// TIA Portal V15.1 export
// export: Created 2024-05-17T05:38:41.6843749Z, ExportSetting WithDefaults, DisplayName Totally Integrated Automation Portal, DisplayVersion V15.1 Update 5, DisplayName TIA Portal Openness, DisplayVersion V15.1 Update 5, DisplayName SINAMICS Startdrive Advanced, DisplayVersion V15.1, DisplayName G130, G150, S120, S150, SINAMICS MV, S210, DisplayVersion V15.1, DisplayName G110M, G120, G120C, G120D, G120P, DisplayVersion V15.1, DisplayName STEP 7 Professional, DisplayVersion V15.1 Update 5, DisplayName STEP 7 Safety, DisplayVersion V15.1, DisplayName WinCC Professional, DisplayVersion V15.1 Update 5, DisplayName SIMATIC Visualization Architect, DisplayVersion V15.1
FUNCTION "LGBHoist2Pos2S-FC302PN-Config" : Void   // FC6606, FBD
TITLE = LMoveEPos-Config / LHoist2Pos2S-FC302PN-Config
{ S7_Optimized_Access := 'FALSE' }
AUTHOR : VCC
FAMILY : Config
VERSION : 0.0.0.0
// =============================================================================
// Configuration MoveUnitEpos
// =============================================================================
// stored: AutoNumber false, IsIECCheckEnabled false, SetENOAutomatically False, UDAEnableTagReadback false
   VAR_INPUT
      C_InitDirection : Bool;   // Config
      C_SafetySwNc : Bool;   // Config
      C_SafetySwUsed : Bool;   // Config
      C_MotorProtectionNc : Bool;   // Config
      C_MotorProtectionUsed : Bool;   // Config
      C_BrakeProtectionNc : Bool;   // Config
      C_BrakeProtectionUsed : Bool;   // Config
      C_ReleaseBrakeUsed : Bool;   // Release brake used / Config
      C_MotionStopUsed : Bool;   // Config
      C_EnableAlarmHW : Bool;   // Enable Alarm hardware (e.g. safetyswitch, motorprotector, detections) / Config
      C_EnablePNReset : Bool;   // Config
      C_NotQuickStop : Bool;   // QuickStop function; When FALSE the QuickStop of the G120 is active / Config
      C_RunTimeMaxSetAlm : DInt;   // Maximum Time (x1ms) that the function may run (create Overtime) / Config
      C_RunTimeMaxResAlm : DInt;   // Maximum Time (x1ms) that the function may run (create Overtime) / Config
      C_HWSubInput : HW_SUBMODULE;   // I/O / Config
      C_HWSubOutput : HW_SUBMODULE;   // I/O / Config
   END_VAR
   VAR_IN_OUT
      IO_Config : "Hoist2Pos2S-FC302PNConfig";   // Output Word / Config
   END_VAR
BEGIN

REGION Network 1: **** 1 - Inputs **** Move Bit Config
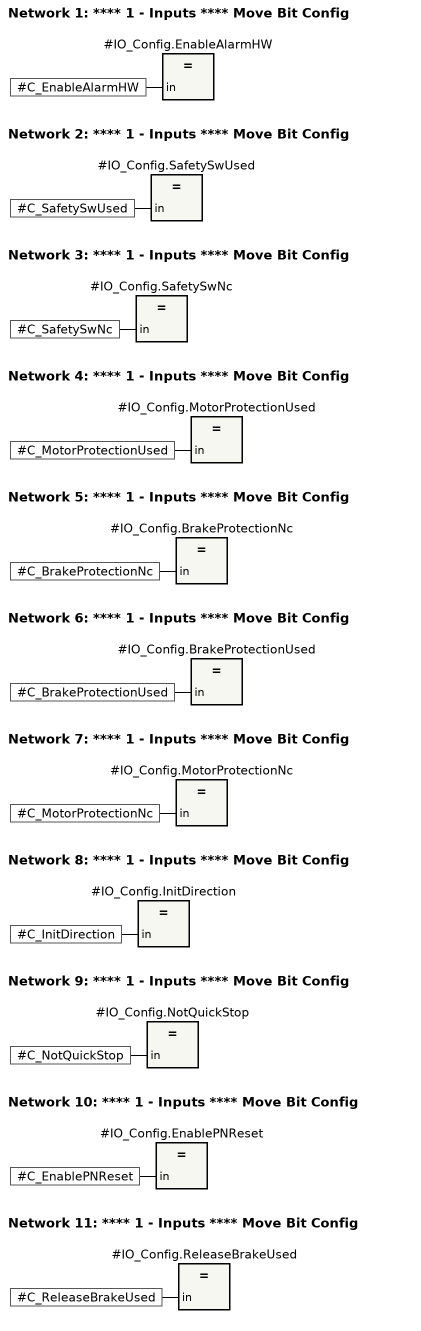
   #IO_Config.EnableAlarmHW := #C_EnableAlarmHW;
END_REGION

REGION Network 2: **** 1 - Inputs **** Move Bit Config
   #IO_Config.SafetySwUsed := #C_SafetySwUsed;
END_REGION

REGION Network 3: **** 1 - Inputs **** Move Bit Config
   #IO_Config.SafetySwNc := #C_SafetySwNc;
END_REGION

REGION Network 4: **** 1 - Inputs **** Move Bit Config
   #IO_Config.MotorProtectionUsed := #C_MotorProtectionUsed;
END_REGION

REGION Network 5: **** 1 - Inputs **** Move Bit Config
   #IO_Config.BrakeProtectionNc := #C_BrakeProtectionNc;
END_REGION

REGION Network 6: **** 1 - Inputs **** Move Bit Config
   #IO_Config.BrakeProtectionUsed := #C_BrakeProtectionUsed;
END_REGION

REGION Network 7: **** 1 - Inputs **** Move Bit Config
   #IO_Config.MotorProtectionNc := #C_MotorProtectionNc;
END_REGION

REGION Network 8: **** 1 - Inputs **** Move Bit Config
   #IO_Config.InitDirection := #C_InitDirection;
END_REGION

REGION Network 9: **** 1 - Inputs **** Move Bit Config
   #IO_Config.NotQuickStop := #C_NotQuickStop;
END_REGION

REGION Network 10: **** 1 - Inputs **** Move Bit Config
   #IO_Config.EnablePNReset := #C_EnablePNReset;
END_REGION

REGION Network 11: **** 1 - Inputs **** Move Bit Config
   #IO_Config.ReleaseBrakeUsed := #C_ReleaseBrakeUsed;
END_REGION

REGION Network 12: **** 1 - Inputs **** Move Bit Config
   // Move Bit Config
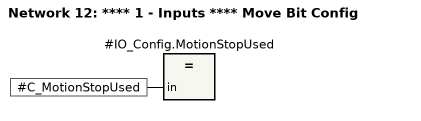
   #IO_Config.MotionStopUsed := #C_MotionStopUsed;
END_REGION

NETWORK
TITLE = **** 1 Inputs **** Move Config UDT
// Move Config
      L     #C_RunTimeMaxSetAlm;
      T     #IO_Config.RunTimeMaxSetAlm;
      L     #C_RunTimeMaxResAlm;
      T     #IO_Config.RunTimeMaxResAlm;
      L     #C_HWSubInput;
      T     #IO_Config.HWSubInput;
      L     #C_HWSubOutput;
      T     #IO_Config.HWSubOutput;

END_FUNCTION
